FUNCTION_BLOCK EventLogger
VAR
    bInit : BOOL := TRUE; 
    bRaise : BOOL := FALSE; 
	bConfirm : BOOL := FALSE; 
	bClear : BOOL := FALSE; 

	newAlarm	: FB_Alarm;
	newWarning	: FB_Alarm;
	event3		: FB_Alarm;
END_VAR


newAlarm(
	Alarm_Event:= TC_EVENTS.WindWings.Encoder_No_Response, 
	bInit:= bInit, 
	bRaise:= bRaise, 
	bConfirm:= bConfirm , 
	bClear:= bClear);


newWarning(
	Alarm_Event:= TC_EVENTS.WindWings.Encoder_Warning, 
	bInit:= bInit, 
	bRaise:= bRaise, 
	bConfirm:= bConfirm , 
	bClear:= bClear);
	
event3(
	Alarm_Event:= TC_EVENTS.WindWings.EventMedNamn3, 
	bInit:= bInit, 
	bRaise:= bRaise, 
	bConfirm:= bConfirm , 
	bClear:= bClear);

	
	bInit := FALSE; 
    bRaise := FALSE; 
	bConfirm := FALSE; 
	bClear := FALSE;

END_FUNCTION_BLOCK

(* stored: Version 1.1.0.1, ProductVersion 3.1.4024.9
   POU EventLogger: Id {276dd7fb-18e2-4dad-96f4-303888d2e089}, SpecialFunc None *)
